TEXTLIST BetrAnzeigeListe
  6 = 'Einzel-Schritt, Litze einführen' | EN: 'Operating mode: Single step,  Steps with Start button, Exit with Single step' | DE: 'Betriebsart: Einzelschritt, Schritte mit Taste START, Beenden mit Einzelschritt' | FR: 'Mode de fonctionnement : Etape individuelle, Etape avec touche Start, Terminer avec étape individuelle' | HU: 'Üzemmód: Egyes lépés,  lépések a Start gombbal,  Befejezés egyes lépéssel' | IT: 'Modalità operativa: Passo-passo,  Avanzare con START, Uscire con Passo-passo' | RU: 'Режим работы: Отдельный шаг,  Шаги с кнопкой Start, ' | RO: 'Mod de operare: pas cu pas \\pasi cu tasta START\\ Iesire din "pas cu pas"' | ES: 'Modo de funcionamiento: Paso individual,  Pasos pulsando Start,  Salir con Paso individual' | PL: 'Tryb pracy: Pojedynczy krok,  Kroki poprzez przyscisk Start, Wyjście poprzez pojedynczy krok' | JA: '作業モード:\u3000シングルステップ, スタートボタンでステップ毎に動作, シングルステップの終了' | ZH: '运行模式: 步进模式, 按启动按钮步进, 通过步进退出'
  7 = 'Einzel-Schritt weiter mit Start' | EN: 'Operating mode: Single step  Steps with Start button Exit with Single step' | DE: 'Betriebsart: Einzelschritt, Schritte mit Taste START, Beenden mit Einzelschritt' | FR: 'Mode de fonctionnement : Etape individuelle Etape avec touche Start Terminer avec étape individuelle' | HU: 'Üzemmód: Egyes lépés  lépések a Start gombbal  Befejezés egyes lépéssel' | IT: 'Modalità operativa: Passo-passo  Avanzare con START Uscire con Passo-passo' | RU: 'Режим работы: Отдельный шаг  Шаги с кнопкой Start ' | RO: 'Mod de operare: pas cu pas \\pasi cu tasta START\\ Iesire din "pas cu pas"' | ES: 'Modo de funcionamiento: Paso individual  Pasos pulsando Start  Salir con Paso individual' | PL: 'Tryb pracy: Pojedynczy krok  Kroki poprzez przyscisk Start Wyjście poprzez pojedynczy krok' | JA: '作業モード:\u3000シングルステップ スタートボタンでステップ毎に動作 シングルステップの終了' | ZH: '运行模式: 步进模式 按启动按钮步进 通过步进退出'
  10 = 'Maschine bereit, Weiter mit Taste START' | EN: 'Machine ready  Continue with START button' | DE: 'Maschine bereit, Weiter mit Taste START' | FR: ' Machine opérationnelle  Continuer avec touche START' | HU: ' Gép készen áll  Tovább a START gombbal' | IT: 'Macchina pronta Premere il tasto START per continuare' | RU: 'Аппарат готов  Продолжить кнопкой START' | RO: 'Masina pregatita\\ Continua cu tasta START' | ES: 'Máquina preparada  Continue pulsando START' | PL: 'Maszyna gotowa  kontynuacja poprzez przycisk START' | JA: '準備完了\\スタートボタンを押してください' | ZH: ' 设备待机  按启动按钮继续'
  11 = 'Maschine bereit zum Crimpen - Litze einführen' | EN: 'Machine ready for crimping   Insert wire' | DE: 'Maschine bereit zum Crimpen, Litze einführen' | FR: 'Machine opérationnelle pour sertissage  Introduire fil' | HU: 'Gép krimpelésre kész  Huzal behelyezése\\' | IT: 'Macchina pronta per crimpare  Inserire il cavo' | RU: 'Машина готова к обжиму  Завести провод' | RO: 'Masina pregatita pentru sertizare\\ Introduceti lita' | ES: 'Máquina preparada para engaste   Insertar cable' | PL: 'Maszyna gotowa do zaciskania   Wprowadzić przewód' | JA: '圧着準備完了 ケーブル挿入' | ZH: '设备待机准备压接   送线'
  12 = 'Maschine im Ablauf gestoppt - Weiter mit START' | EN: 'Machine stopped during process  Continue with START' | DE: 'Maschine im Ablauf gestoppt, Weiter mit START' | FR: ' Machine arrêtée en cours  Continuer avec touche START' | HU: ' Gép a folyamat közben megállítva  Tovább a START-tal' | IT: 'La macchina si è bloccata durante il processo Premere START per continuare' | RU: 'Остановка машины во время работы  Продолжить кнопкой START' | RO: 'Masina s-a oprit in timpul procesului\\ Continua cu tasta START' | ES: 'Máquina parada durante el proceso  Continue con START' | PL: 'Maszyna zatrzymana w czasie procesu  kontynuacja poprzez przycisk START' | JA: '機械が動作中停止しました スタートボタンを押してください' | ZH: ' 运行中设备停止  按启动按钮继续'
  13 = 'nicht Crimpen zu (?)' | EN: 'Open crimping tool for setup Close with Start button Exit with Reset' | DE: 'Crimpzange zum Einrichten offen, Schließen mit Taste Start, Beenden mit Reset' | FR: 'Ouvrir pince à sertir pour réglage Fermer avec touche Start Terminer avec Reset' | HU: 'Krimpelo fogó beállításhoz nyitva  Zárás a Start gombbal  Befejezés a Reset gombbal' | IT: 'Apertura ganasce di crimpatura per regolazione Chiusura con pulsante START Uscire con RESET' | RU: 'Открыть обжимной элемент для настройки   Закрыть кнопкой Start  Выход через Reset' | RO: 'Cleste crimpare deschis pentru reglare\\ Inchidere cu tasta START\\ Incheiere cu tasta RESET' | ES: 'Herramienta de crimpado abierta para ajuste Cerrar pulsando Start Salir pulsando Reset' | PL: 'Otwarcie jednostki zaciskającej do ustawienia Zamknięcie poprzez przycisk Start Wyjście poprzez przycisk Reset' | JA: 'セットアップ時の圧着ツールオープン スタートボタンでクローズ/nリセッットで終了' | ZH: '打开压接工具来设定 按启动按钮关闭 按复位按钮退出'
  14 = 'Crimpen zu (?)' | EN: 'Crimping tool closed for testing Open with Start button Exit with Reset' | DE: 'Crimpzange zum Prüfen zu Öffnen mit Taste Start, Beenden mit Reset' | FR: 'Fermer pince à sertir pour contrôle Ouvrir avec touche Start Terminer avec Reset' | HU: 'Krimpelo fogó ellenorzéshez zárva  Nyitás a Start gombbal  Befejezés a Reset gombbal' | IT: 'Ganasce di crimpatura chiuse per test Aprire con pulsante START Uscire con RESET' | RU: 'Обжимной элемент закрыт для теста  Открыть кнопкой Старт Завершить с помощью Reset' | RO: 'Cleste crimpare inchis pentru verificare\\ deschidere cu tasta START\\ Incheiere  cu tasta RESET' | ES: 'Herramienta de crimpado cerrada para ajuste Abrir pulsando Start Salir pulsando Reset' | PL: 'Jednostka zaciskająca zamknięta do testowania Otwarcie maszyny poprzez przycisk Wyjście poprzez przycisk Reset' | JA: 'テスト時の圧着ツールクローズ スタートボタンでオープン リセットで終了' | ZH: '关闭压接工具来测试 按启动按钮开机 按复位按钮退出'
  15 = 'Bereit zum Crimpen - Litze einführen-dann Start drücken' | EN: 'Machine ready for crimping  Insert wire and press Start button' | DE: 'Maschine bereit zum Crimpen, Litze einführen und Taste Start drücken' | FR: 'Machine opérationnelle pour sertissage  Introduire fil et appuyer touche Start' | HU: 'Gép krimpelésre kész  Huzal behelyezése\\ és  nyomja meg a Start gombot' | IT: 'Macchina pronta per crimpare Inserire il cavo e premere il pulsante START' | RU: 'Машина готова к обжиму  Завести провод и  нажать кнопку Старт' | RO: 'Masina pregatita pentru sertizare\\ Introduceti lita si \\ apasa tasta START' | ES: 'Máquina preparada para engaste  Insertar cable y pulsar Start' | PL: 'Maszyna gotowa do zaciskania  Wprowadzić przewód i  nacisnąć przycisk Start' | JA: '圧着準備完了 ケーブル挿入 スタートボタンを押してください' | ZH: '设备待机准备压接  送线  按下启动按钮'
  20 = 'Abisolieren einrichten - weiter mit Start' | EN: 'Operating mode:  Set up stripping unit Continue with Start Exit with Reset' | DE: 'Betriebsart: Abisolieren einrichten, weiter mit Start, Beenden mit Reset' | FR: 'Mode de fonctionnement :  Régler dénudage Continuer avec Start Terminer avec Reset' | HU: 'Üzemmód:  Csupaszítás beállítása  tovább a Start gombbal Befejezés a Reset gombbal' | IT: 'Modalità operativa: Impostazione unità di spellatura Continuare con START Uscire con RESET' | RU: 'Режим работы: Настройка снятия изоляции  Продолжить с Start Выход с Reset' | RO: 'Mod de operare: reglare dezizolare\\continua cu tasta START\\ Incheiere cu RESET' | ES: 'Modo de funcionamiento: Ajustar unidad de pelado Continuar con Start Salir con Reset' | PL: 'Tryb pracy: Ustawianie jednostki zaciskającej Kontynuacja poprzez przycisk Start Wyjście poprzez przycisk Reset' | JA: '作業モード:\u3000ストリッピング・ユニットのセットアップ スタートして継続/リセットして終了' | ZH: '运行模式: 设定剥线单元  按启动按钮继续 通过复位退出 '
  21 = 'Magazin Leerfahren (?)' | EN: 'Operating mode:  Run magazine empty Exit with Reset' | DE: 'Betriebsart: Magazin leerfahren, Beenden mit Reset' | FR: 'Mode de fonctionnement :  Vider magasin Terminer avec Reset' | HU: 'Üzemmód:  Tároló üresre járatása Befejezés a Reset gombbal' | IT: 'Modalità operativa:  Svuotamento caricatore Uscire con RESET' | RU: 'Вид операции:  Очистить магазин Завершить с помощью Reset' | RO: 'Mod de operare: \\ golire magazie \\ Incheiere  cu tasta RESET' | ES: 'Modo de funcionamiento:  Ejecutar vaciado de depósito Salir con Reset' | PL: 'Tryb pracy:   Uruchomienie pustego magazynka Wyjście poprzez przycisk Reset' | JA: '作業モード:\u3000 マガジンが空の状態での操作 リセットで終了' | ZH: '运行模式:   启动料箱清空 通过复位退出 '
  22 = 'Sortierer Leerfahren (?)' | EN: 'Operating mode:  Run sorter empty Exit with Reset' | DE: 'Betriebsart: Sortierer leerfahren, Beenden mit Reset' | FR: 'Mode de fonctionnement :  Vider trieuse Terminer avec Reset' | HU: 'Üzemmód:  Szortírozó üresre járatása Befejezés a Reset gombbal' | IT: 'Modalità operativa: Scarico canale contatti Uscire con RESET' | RU: 'Вид операции:  Очистка сортировщика Завершить с помощью Reset' | RO: 'Mod de operare: \\ golire sortator \\ Incheiere  cu tasta RESET' | ES: 'Modo de funcionamiento:  Ejecutar vaciado clasificador Salir con Reset' | PL: 'Tryb pracy:   Uruchomienie pustego sortera Wyjście poprzez przycisk Reset' | JA: '作業モード:\u3000 ソーター空状態での操作 リセットで終了' | ZH: '运行模式:   运行分拣清空 通过复位退出 '
  23 = 'Crimpen Einrichten (?)' | EN: 'Operating mode:  Set up crimping Exit with Reset' | DE: 'Betriebsart: Crimpzange einrichten, Beenden mit Reset' | FR: 'Mode de fonctionnement :  Régler pince à sertir Terminer avec Reset' | HU: 'Üzemmód:  Krimpelo fogó beállítása Befejezés a Reset gombbal' | IT: 'Modalità operativa:  Regolazione crimpatura Uscire con RESET' | RU: 'Вид операции:  Настройка обжимного элемента Завершить с помощью Reset' | RO: 'Mod de operare: \\ reglare cleste sertizare\\ Incheiere cu tasta RESET' | ES: 'Modo de funcionamiento:  Ajustar engaste Salir con Reset' | PL: 'Tryb pracy:   Ustawienie zaciskania Wyjście poprzez przycisk Reset' | JA: '作業モード:\u3000 圧着の設定 リセットで終了' | ZH: '运行模式:   设定压接 通过复位退出 '
  24 = 'Abisolieren einrichten - Litze einführen' | EN: 'Operating mode:  Set up stripping unit Insert wire Exit with Reset' | DE: 'Betriebsart: Abisolieren einrichten, Litze einführen, Beenden mit Reset' | FR: 'Mode de fonctionnement :  Régler dénudage Introduire fil Terminer avec Reset' | HU: 'Üzemmód:  Csupaszítás beállítása Huzal behelyezése Befejezés a Reset gombbal' | IT: 'Modalità operativa: Impostazione unità di spellatura Inserire il cavo Uscire con RESET' | RU: 'Режим работы: Настройка снятия изоляции  завести провод Выход с Reset' | RO: 'Mod de operare: reglare dezizolare\\ introducere lita\\ Incheiere cu RESET' | ES: 'Modo de funcionamiento: Ajustar unidad de pelado Insertar cable Salir con Reset' | PL: 'Tryb pracy: Ustawianie jednostki zaciskającej Wprowadzić przewód Wyjście poprzez przycisk Reset' | JA: '作業モード:\u3000ストリッピング・ユニットのセットアップ ケーブルの挿入/リセットして終了' | ZH: '运行模式: 设定剥线单元   送线   通过复位退出 '
  25 = 'Probelauf ohne Kontakt' | EN: 'Operating mode:  Trial run without contact Exit with Reset' | DE: 'Betriebsart: Probelauf ohne Kontakt, Beenden mit Reset' | FR: "Mode de fonctionnement :  Marche d'essai sans contact Terminer avec Reset" | HU: 'Üzemmód:  Próbaüzem érintkezo nélkül Befejezés a Reset gombbal' | IT: 'Modalità operativa: Ciclo di prova senza contatto Uscire con RESET' | RU: 'Вид операции:  Пробный запуск без контактов Завершить с помощью Reset' | RO: 'Mod de operare: \\ test fara contacte \\ Incheiere  cu tasta RESET' | ES: 'Modo de funcionamiento:  Prueba sin contacto  Salir con Reset' | PL: 'Tryb pracy:   Przebieg testowy bez kontaktu Wyjście poprzez przycisk Reset' | JA: '作業モード:\u3000 コンタクトなしでのテスト操作 リセットで終了' | ZH: '运行模式:   试运行但不进针 通过复位退出 '
  26 = 'Probelauf ohne Crimpen' | EN: 'Operating mode:  Trial run without crimping Exit with Reset' | DE: 'Betriebsart: Probelauf ohne Crimpen, Beenden mit Reset' | FR: "Mode de fonctionnement :  Marche d'essai sans sertissage Terminer avec Reset" | HU: 'Üzemmód:  Próbaüzem krimplelés nélkül Befejezés a Reset gombbal' | IT: 'Modalità operativa: Ciclo di prova senza crimpatura Uscire con RESET' | RU: 'Вид операции:  Пробный запуск без обжима Завершить с помощью Reset' | RO: 'Mod de operare: \\ test fara sertizare \\ Incheiere  cu tasta RESET' | ES: 'Modo de funcionamiento:  Prueba sin engaste  Salir con Reset' | PL: 'Tryb pracy:   Przebieg testowy bez zaciskania Wyjście poprzez przycisk Reset' | JA: '作業モード:\u3000 圧着なしでのテスト操作 リセットで終了' | ZH: '运行模式:   试运行但不压接 通过复位退出 '
  27 = 'Probelauf ohne Litze' | EN: 'Operating mode:  Trial run without wire Exit with Reset' | DE: 'Betriebsart: Probelauf ohne Litze Beenden, mit Reset' | FR: "Mode de fonctionnement :  Marche d'essai sans fil Terminer avec Reset" | HU: 'Üzemmód:  Próbaüzem huzal nélkül Befejezés a Reset gombbal' | IT: 'Modalità operativa: Ciclo di prova senza cavo Uscire con RESET' | RU: 'Вид операции:  Пробный запуск без кабеля Завершить с помощью Reset' | RO: 'Mod de operare: \\ test fara lite \\ Incheiere cu tasta RESET' | ES: 'Modo de funcionamiento:  Prueba sin cable  Salir con Reset' | PL: 'Tryb pracy:   Przebieg testowy bez przewodu Wyjście poprzez przycisk Reset' | JA: '作業モード:\u3000 ケーブルなしでのテスト操作 リセットで終了' | ZH: '运行模式:   试运行但不进线 通过复位退出 '
  55 = 'A55 Kontakt nicht gefallen' | EN: 'Malfunction: Contact not fed E1.10 missing' | DE: 'Störung: Kontakt nicht gefallen E1.10 fehlt' | FR: 'Défaut : contact pas tombé E1.10 absent' | HU: 'Zavar: Érintkezo nem esett le E1.10 hiányzik' | IT: 'Anomalia: Contatto non in posizione E1.10 mancante' | RU: 'Нарушение: Контакт не загружен, E1.10 отсутствует' | RO: 'Defectiune: Contactul nu a cazut\\ E1.10 lipseste' | ES: 'Error de funcionamiento: Contactos no alimentados E1.10 sin señal' | PL: 'Nieprawidłowość:  Kontakt niepodany E1.10 Brakuje' | JA: 'エラー: コンタクトが供給されていません E1.10\u3000不明' | ZH: '故障: 针没有落下 E1.10 故障'
  1000 = 'ohne Sortierluft' | EN: 'without sorting air' | DE: 'ohne Sortierluft' | FR: "sans tri d'air" | HU: 'buborékok nélkül' | IT: 'senza aria' | RU: 'без пузырьков' | RO: 'fără bule' | ES: 'sin burbujas' | PL: 'bez bąbelków' | JA: '空気をソートせずに' | ZH: '没有分拣气'
  1001 = 'mit Sortierluft' | EN: 'with sorting air' | DE: 'mit Sortierluft' | FR: "avec tri de l'air" | HU: 'buborékokkal' | IT: 'con aria' | RU: 'с пузырьками' | RO: 'cu bule' | ES: 'con burbujas' | PL: 'z bąbelkami' | JA: 'ソートエアー付き' | ZH: '带分拣气'
  127 = 'warte auf SAFETY-Signal...'
  101 = 'Druckluft nicht ein'
  102 = 'Schutztür nicht zu'
  105 = 'Kein Signal von Taste Maschine-Aus'
  108 = 'Not-Aus Steuerpult nicht OK'
  109 = 'Kein SAFETY Signal'
  501 = 'Fehler: A1.8 "Kontakt schieben" ist aus, aber Schieber ist vorn.'
  502 = 'Fehler: A1.8 "Kontakt schieben" ist ein, aber Schieber ist nicht vorn.'
  503 = 'Fehler: A1.9 "Crimpeinheit vor" ist aus, Einheit ist aber nicht hinten.'
  504 = 'Fehler: A1.9 "Crimpeinheit vor" ist ein, Einheit ist aber nicht vorn.'
  505 = 'Fehler: A1.10 "Abisolierer nach links" ist aus, aber Einheit ist links.'
  506 = 'Fehler: A1.10 "Abisolierer nach links" ist ein, aber Einheit ist nicht links.'
  507 = 'Fehler: A1.11 "Abisolierer zu" ist aus, aber Abisolierer ist zu.'
  508 = 'Fehler: A1.11 "Abisolierer zu" ist ein, aber Abisolierer ist nicht zu.'
  509 = 'Fehler A1.13 "Abisolierer zurück" ist aus, aber Abisolierer ist nicht vorn.'
  510 = 'Fehler A1.13 "Abisolierer zurück" ist ein, aber Abisolierer ist nicht hinten.'
  511 = 'Fehler A1.14 "Crimpzange zu" ist aus, aber Zange ist nicht offen.'
  512 = 'Fehler A1.14 "Crimpzange zu" ist ein, aber Zange ist offen.'
  513 = 'Fehler A1.15 "Drahthalter zu" ist aus, aber Drahthalter ist nicht offen.'
  514 = 'Fehler A1.15 "Drahthalter zu" ist ein, aber Drahthalter ist offen.'
  500 = '   '
  420 = 'Einzelschritt - Start durch Drahteinfuhr'
  422 = 'Abisolierer zu'
  423 = 'Abisolierer zurück (abisolieren)'
  424 = 'Abisolierer nach links + Abisolierer auf'
  425 = 'Crimpeinheit vor'
  426 = 'Crimpen zu'
  427 = 'Drahthalter + Drahtführung auf'
  428 = 'Crimpzange auf + Abisoliereinheit vor'
  429 = 'Ausstoßen vor'
  430 = 'Crimpeinheit zurück'
  431 = 'Abisolierer nach rechts + Kontakt-Schieben zurück'
  432 = 'Einzelschritt - Ende'
  421 = 'Drahthalter + Drahtführung zu'
  600 = 'Störung: Drahthalter nicht offen, E1.2 fehlt' | EN: 'Malfunction: Wire holder not open, E1.2 missing' | DE: 'Störung: Drahthalter nicht offen, E1.2 fehlt' | FR: 'Défaut : Porte-fil pas ouvert, E1.2 absent' | HU: 'Zavar: Huzaltartó nincs nyitva, E1.2 hiányzik' | IT: 'Anomalia: Dispositivo blocca-cavo chiuso, E1.2 mancante' | RU: 'Нарушение: Кабельный захват не открыт, E1.2 отсутствует' | RO: 'Defectiune: Suportul de fir nu e deschis, E1.2 lipseste' | ES: 'Error de funcion.: Soporte de cable no está abierto, E1.2 sin señal' | PL: 'Nieprawidłowość: Uchwyt przewodu nie jest otwarty, E1.2 Brakuje' | JA: 'エラー: ケーブルフォルダーが閉じていません, E1.2 不明' | ZH: '故障: 集线器未打开, E1.2 缺失'
  601 = 'Störung: Drahthalter nicht zu E1.2 nicht weg' | EN: 'Malfunction: Wire holder not closed, E1.2 not gone' | DE: 'Störung: Drahthalter nicht zu, E1.2 nicht weg' | FR: 'Défaut : Porte-fil pas fermé, E1.2 pas parti' | HU: 'Zavar: Huzaltartó nincs zárva, E1.2 nem tunt el' | IT: 'Anomalia: Dispositivo blocca-cavo aperto, E1.2 non attivo' | RU: 'Нарушение: Кабельный захват не закрыт, E1.2 не удален' | RO: 'Defectiune: Suportul de fir nu e inchis, E1.2 nu dispare' | ES: 'Error de funcion.: Soporte de cable no está cerrado, E1.2 no desaparece la señal' | PL: 'Nieprawidłowość: Uchwyt przewodu nie jest zamknięty, E1.2 Pozostaje' | JA: 'エラー: ワイヤーホルダーが閉じていません, E1.2 不明' | ZH: '故障: 集线器未关闭, E1.2 没有离开'
  602 = 'Störung: Auslöseschalter Dauermeldung E1.3 nicht weg' | EN: 'Malfunction: Cable trigger switch continuous signal, E1.3 not gone' | DE: 'Störung: Auslöseschalter Dauermeldung, E1.3 nicht weg' | FR: 'Défaut : Déclencheur message permanent, E1.3 pas parti' | HU: 'Zavar: Kioldó kapcsoló folyamatos jelzés, E1.3 nem tunt el' | IT: 'Anomalia: Segnale continuo del sensore di presenza cavo, E1.3 non attivo' | RU: 'Нарушение: Непрерывный сигнал блокировки, E1.3 не удален' | RO: 'Defectiune: Declanșator mesaj permanent, E1.3 nu dispare' | ES: 'Error de funcion.: Señal permanente en interruptor de disparo de cable, E1.3 no desaparece' | PL: 'Nieprawidłowość: Przełącznik kablowy z ciągłym sygnałem, E.1.3 Pozostało' | JA: 'エラー: ケーブルトリガースイッチが連続メッセージ, E1.3\u3000未完了' | ZH: '故障:线缆触发开关持续信号, E1.3 故障没有解除'
  603 = 'Störung: Abisoliermesser nicht offen E1.4 nicht weg' | EN: 'Malfunction: Stripping blades not open, E1.4 not gone' | DE: 'Störung: Abisoliermesser nicht offen, E1.4 nicht weg' | FR: 'Défaut : Lames à dénuder pas ouvertes, E1.4 pas parti' | HU: 'Zavar: Csupaszító kés nincs nyitva, E1.4 nem  tunt el' | IT: 'Anomalia: Lame di spellatura non aperte, E1.4 non attivo' | RU: 'Нарушение: Нож зачистки не открыт, E1.4 не удален' | RO: 'Defectiune: Cutitul de dezizolare nu e deschis, E1.4 nu dispare' | ES: 'Error de funcion.: Cuchillas de pelado no abiertas, E1.4 no desaparece la señal' | PL: 'Nieprawidłowość:  Noże odizolowujące nie są otwarte, E1.4 Pozostało' | JA: 'エラー: ストリッピングブレードが開いていません,  E1.4\u3000未完了' | ZH: '故障: 剥线刀片没有打开, E1.4 故障没有解除'
  604 = 'Störung: Abisoliermesser nicht  zu E1.4 fehlt' | EN: 'Malfunction: Stripping blades not closed, E1.4 missing' | DE: 'Störung: Abisoliermesser nicht  zu, E1.4 fehlt' | FR: 'Défaut : Lames à dénuder pas fermées, E1.4 absent' | HU: 'Zavar: Csupaszító kés nincs zárva, E1.4 hiányzik' | IT: 'Anomalia: Lame di spellatura non chiuse, E1.2 mancante' | RU: 'Нарушение: Нож зачистки не закрыт, E1.4 отсутствует' | RO: 'Defectiune: Cutitul de dezizolare nu e inchis, E1.4 lipseste' | ES: 'Error de funcion.: Cuchillas de pelado no cerradas, E1.4 sin señal' | PL: 'Nieprawidłowość: Nnoże odizolowujące nie są zamknięte, E1.4 Brakuje' | JA: 'エラー: ストリッピングブレードが閉じていません, 1.4不明' | ZH: '故障: 剥线刀片没有闭合 E1.4 故障'
  605 = 'Störung: Doppelmeldung Abisolierer vorn+rück E1.5+E1.6 gleichzeitig' | EN: 'Malfunction: Double signal stripping unit at front+rear E1.5+E1.6 simultaneous' | DE: 'Störung: Doppelmeldung Abisolierer vorn+rück, E1.5+E1.6 gleichzeitig' | FR: 'Défaut : Message double Dénudeur avance+retour, E1.5+E1.5 simultanément' | HU: 'Zavar: Dupla jelzés Csupaszító elol+vissza, E1.5+E1.6 egyszerre' | IT: 'Anomalia: Segnale doppio Unità di spellatura avanzata+arretrata E1.5+E1.6 contemporaneamente' | RU: 'Нарушение: Двухкратное сообщение блок зачистки фронтальный + задней панелиnE1.3+E1.4 одновременно' | RO: 'Defectiune: Mesaj dublu dezizolator inainte+inapoi, E1.5+E1.6 simultan' | ES: 'Error de funcion.: Doble señal la unidad de pelado está delante y detrás E1.3+E1.4 simultaneamente' | PL: 'Nieprawidłowość: Podwójny sygnał jednostka odizolowująca z przodu+tyłu E1.3+E1.4 Równocześnie' | JA: 'エラー:ダブルメッセージ ストリッピングユニットが前面+後方にあります E2.1+E2.4\u3000同時発生' | ZH: '故障:    双路信号 剥线单元在前+在后 E1.3+E1.4 同时'
  606 = 'Störung: Abisolierer nicht vorn E1.5 fehlt' | EN: 'Malfunction: Stripping unit not at front, E1.5 missing' | DE: 'Störung: Abisolierer nicht vorn, E1.5 fehlt' | FR: 'Défaut : Dénudeur pas avance, E1.5 absent' | HU: 'Zavar: Csupaszító kés nincs elöl, E1.5 hiányzik' | IT: 'Anomalia: Unità di spellatura non avanzata, E1.5 mancante' | RU: 'Нарушение: Зачистка не фронтально, E1.5 отсутствует' | RO: 'Defectiune: Dezizolatorul nu e in fata, E1.5 lipseste' | ES: 'Error de funcion.: La unidad de pelado no está en la parte frontal, E1.3 sin señal' | PL: 'Nieprawidłowość: Jednostka odizolowująca nie jest z przodu, E1.5 Brakuje' | JA: 'エラー: ストリッピングユニットが前面に有りません, E1.5\u3000不明' | ZH: '故障: 剥线单元不在前边, E1.5 故障'
  607 = 'Störung: Abisolierer nicht rück (abisoliert) E1.6 fehlt' | EN: 'Malfunction: Stripping unit not at rear (stripped),  E1.6 missing' | DE: 'Störung: Abisolierer nicht rück (abisoliert),  E1.6 fehlt' | FR: 'Défaut : Dénudeur pas retour (dénudé),  E1.6 absent' | HU: 'Zavar: Csupaszító nincs hátul (csupaszított), E1.6 hiányzik' | IT: 'Anomalia: Unità si spellatura non arretrata (spellato), E1.6 mancante' | RU: 'Нарушение: Зачистка не с тыльной стороны (зачистка), E1.6 отсутствует' | RO: 'Defectiune: Dezizolatorul nu revine in spate, E1.6 lipseste' | ES: 'Error de funcion.: La unidad de pelado no está en la parte posterior (despojado), E1.6 sin señal' | PL: 'Nieprawidłowość: Jednostka odizolowująca nie jest z tyłu (odizolowane), E1.6 Brakuje' | JA: 'エラー: ストリッピングユニットが後方に有りません （除去済み), E1.6 不明' | ZH: '故障: 剥线单元不在后边 (剥离), E1.6 故障'
  608 = 'Störung: Abisolierer nicht links (aus Arbeitsraum) E1.7 fehlt' | EN: 'Malfunction: Stripping unit not on LH side (out of machining compartment), E1.7 missing' | DE: 'Störung: Abisolierer nicht links (aus Arbeitsraum), E1.7 fehlt' | FR: "Défaut : Dénudeur pas gauche (de l'espace de travail), E1.7 absent" | HU: 'Zavar: Csupaszító nincs bal oldalon (a munkatérbol), E1.7 hiányzik' | IT: 'Anomalia: Unità di spellatura non sul lato LH (fuori dal comparto di lavoro), E1.7 mancante' | RU: 'Нарушение: Блокзачистки не с лева (вне машинного блока), E1.7 отсутствует' | RO: 'Defectiune: Dezizolatorul nu e in stanga (din domeniul de lucru), E1.7 lipseste' | ES: 'Error de funcion.: La unidad de pelado no está en el lado LH (fuera del espacio de trabajo), E1.7 sin señal' | PL: 'Nieprawidłowość: Jednostka odizolowująca nie jest z lewej strony (poza przedziałem maszyny), E1.7 Brakuje' | JA: 'エラー: ストリッピングユニットがLH側に有りません (正しくセットされていません）E1.7 不明' | ZH: '故障: 剥线单元不在左边 ( 不在工作区间 )  E1.7 故障'
  609 = 'Störung: Abisolierer nicht rechts E1.7 nicht weg' | EN: 'Malfunction: Stripping unit not on RH side, E1.7 not gone' | DE: 'Störung: Abisolierer nicht rechts, E1.7 nicht weg' | FR: 'Défaut : Dénudeur pas droite, E1.7 pas parti' | HU: 'Zavar: Huzaltartó nincs jobb oldalon, E1.7 nem tunt el' | IT: 'Anomalia: Unità di spellatura non sul lato RH, E1.7 non attivo' | RU: 'Нарушение: Блокзачистки не с права, E1.7 не удален' | RO: 'Defectiune: Dezizolatorul nu e in dreapta, E1.7 nu dispare' | ES: 'Error de funcionamiento: La unidad de pelado no está en el lado RH, E1.7 no desaparece la señal' | PL: 'Nieprawidłowość: Jednostka odizolowująca nie jest po prawej stronie, E1.7 Pozostało' | JA: 'エラー: ストリッピングユニットがRH側に有りません E1.5\u3000未完了' | ZH: '故障: 剥线单元不在右边, E1.7 故障没有解除'
  610 = 'Störung: Doppelmeldung Crimpzange zu+offen E1.8+E1.9 gleichzeitig' | EN: 'Malfunction: Double signal Crimping tool closed+open, E1.8+E1.9 simultaneous' | DE: 'Störung: Doppelmeldung Crimpzange zu+offen E1.8+E1.9 gleichzeitig' | FR: 'Défaut : Message double Pince à sertir fermée+ouverte E1.8+E1.9 simultanément' | HU: 'Zavar: Dupla jelzés Krimpelo fogó zárva+nyitva, E1.8+E1.9 egyszerre' | IT: 'Anomalia: Segnale doppio Ganasce di crimpatura chiuse+aperte, E1.8+E1.9 contemporaneamente' | RU: 'Нарушение: Двухкратное сообщение обжимной элемент закрать + открыть, E1.8+E1.9 одновременно' | RO: 'Defectiune: Mesaj dublu cleste sertizare inchis+deschis, E1.8+E1.9 simultan' | ES: 'Error de funcionamiento: Doble señal la unidad de crimpado está abierta y cerrada, E1.8+E1.9 simultaneamente' | PL: 'Nieprawidłowość: Podwójny sygnał Jednostka zaciskająca zamknięta+otwarta, E1.8+E1.9 Równocześnie' | JA: 'エラー:ダブルメッセージ ストリッピングユニット\u3000クローズ+オープン E1.8+E1.9 同時発生' | ZH: '故障:   双路信号 压接工具闭合+打开 E1.8+E1.9 同时'
  611 = 'Störung: Crimpzange nicht zu E1.8 fehlt' | EN: 'Malfunction: Crimping tool not closed, E1.8 missing' | DE: 'Störung: Crimpzange nicht zu, E1.8 fehlt' | FR: 'Défaut : Pince à sertir pas fermée, E1.8 absent' | HU: 'Zavar: Csupaszító kés nincs zárva E1.8 hiányzik' | IT: 'Anomalia: Ganasce di crimpatura aperte, E1.8 mancante' | RU: 'Нарушение: Обжимной элемент не закрыт, E1.8 отсутствует' | RO: 'Defectiune: Clestele de sertizare nu e inchis, E1.8 lipseste' | ES: 'Error de funcionamiento: Herramienta de engaste no está cerrada, E1.8 sin señal' | PL: 'Nieprawidłowość: Jednostka zaciskająca nie jest zamknięta, E1.8 Brakuje' | JA: 'エラー: 圧着ツールが閉じていませんE1.8\u3000不明' | ZH: '故障: 压接工具没有关闭, E1.8 故障'
  612 = 'Störung: Crimpzange nicht offen E1.7 fehlt' | EN: 'Malfunction: Crimping tool not open, E1.9 missing' | DE: 'Störung: Crimpzange nicht offen, E1.9 fehlt' | FR: 'Défaut : Pince à sertir pas ouverte, E1.9 absent' | HU: 'Zavar: Csupaszító kés nincs nyitva E1.9 hiányzik' | IT: 'Anomalia: Ganasce di crimpatura chiuse E1.9 mancante' | RU: 'Нарушение: Обжимной элемент не открыт, E1.9 отсутствует' | RO: 'Defectiune: Clestele de sertizare nu e deschis, E1.9 lipseste' | ES: 'Error de funcionamiento: Herramienta de engaste no está abierta, E1.9 sin señal' | PL: 'Nieprawidłowość: Jednostka zaciskająca nie jest otwarta, E1.9 Brakuje' | JA: 'エラー: 圧着ユニットが開いていません, E1.9 不明' | ZH: '故障: 压接工具没有打开, E1.9 故障'
  613 = 'Störung: Kontakt nicht gefallen E1.10 fehlt' | EN: 'Malfunction: Contact not fed, E1.10 missing' | DE: 'Störung: Kontakt nicht gefallen, E1.10 fehlt' | FR: 'Défaut : Contact pas tombé, E1.10 absent' | HU: 'Zavar: Érintkezo nem esett le, E1.10 hiányzik' | IT: 'Anomalia: Contatto non in posizione E1.10 mancante' | RU: 'Нарушение: Контакт не загружен, E1.10 отсутствует' | RO: 'Defectiune: Contactul nu a cazut E1.10 lipseste' | ES: 'Error de funcion.: Contactos no alimentados, E1.10 sin señal' | PL: 'Nieprawidłowość: Kontakt niepodany, E1.10 Brakuje' | JA: 'エラー: コンタクトが供給されていません 1.10\u3000不明' | ZH: '故障: 针没有落下 E1.10 故障'
  614 = 'Störung: Dauermeldung Kontakt gefallen E1.10 nicht weg' | EN: 'Malfunction: Continuous signal, contact fed, E1.10 not gone' | DE: 'Störung: Dauermeldung Kontakt gefallen, E1.10 nicht weg' | FR: 'Défaut : Message permanent contact tombé, E1.10 pas parti' | HU: 'Zavar: Folyamatos jelzés érintkezo leesett, E1.10 nem tunt el' | IT: 'Anomalia: Segnale continuo alimentatore dei contatti, E1.10 non attivo' | RU: 'Нарушение: Непрерывный сигнал контакт не загружен, E1.10 не удален' | RO: 'Defectiune: Mesaj permanent contact cazut, E1.10 nu dispare' | ES: 'Error de funcionamiento: Señal permanente alimentador contactos, E1.10 no desaparece la señal' | PL: 'Nieprawidłowość: Ciągły sygnał, podajnik kontaktów E1.10 Pozostaje' | JA: 'エラー: 連続メッセージ,コンタクト供給, E1.10 未完了' | ZH: '故障: 持续信号，送针, E1.10 故障没有解除'
  615 = 'Störung: Doppelmeldung Crimpeinheit vorn+rück E1.11+E1.12 gleichzeitig' | EN: 'Malfunction:  Double signal Crimping unit at front+rear, E1.11+E1.12 simultaneous' | DE: 'Störung: Doppelmeldung Crimpeinheit vorn+rück, E1.11+E1.12 gleichzeitig' | FR: 'Défaut : Message double Unité à dénuder avance+retour, E1.11+E1.12 simultanément' | HU: 'Zavar:  Dupla jelzés Krimpelo egység elöl+hátul, E1.11+E1.12 egyszerre' | IT: 'Anomalia: Segnale doppio Unità di crimpatura avanzata+arretrata, E1.11+E1.12 contemporaneamente' | RU: 'Нарушение: Двухкратное сообщение Обжимной элемент фронтальный+задний, E1.11+E1.12  одновременно' | RO: 'Defectiune: mesaj dublu unitate sertizare inainte+inapoi E1.11+E1.12 simultan' | ES: 'Error de funcionamiento: Doble señal la unidad de crimpado está delante y detrás E1.11+E1.12 simultaneamente' | PL: 'Nieprawidłowość: Podwójny sygnał Jednostka zaciskająca z przodu+tyłu, E1.11+E1.12 Równocześnie' | JA: 'エラー:ダブルメッセージ 圧着ユニットが前面+後方にありません E1.11+E1.12 同時発生' | ZH: '故障:  双路信号 压接单元 在前+在后 E1.11+E1.12 同时'
  616 = 'Störung: Crimpeinheit nicht vorn E1.11 fehlt' | EN: 'Malfunction: Crimping unit not at front, E1.11 missing' | DE: 'Störung: Crimpeinheit nicht vorn, E1.11 fehlt' | FR: 'Défaut : Unité à dénuder pas avance, E1.11 absent' | HU: 'Zavar: Krimpelo egység nincs elöl, E1.11 hiányzik' | IT: 'Anomalia: Unità di crimpatura non avanzata, E1.11 mancante' | RU: 'Нарушение: Обжимной элемент не фронтально, E1.11 отсутствует' | RO: 'Defectiune: Unitatea de sertizare nu e in fata, E1.11 lipseste' | ES: 'Error de funcionamiento: Unidad de engaste no está en la parte frontal, E1.11 sin señal' | PL: 'Nieprawidłowość: Jednostka zaciskająca nie jest z przodu, E1.11 Brakuje' | JA: 'エラー: 圧着ユニットが前面に有りません,E1.11 不明' | ZH: '故障: 压接单元不在前面 E1.11 故障'
  617 = 'Störung: Crimpeinheit nicht rück E1.12 fehlt' | EN: 'Malfunction: Crimping unit not at rear, E1.12 missing' | DE: 'Störung: Crimpeinheit nicht rück, E1.12 fehlt' | FR: 'Défaut : Unité à dénuder pas retour, E1.12 absent' | HU: 'Zavar: Krimpelo egység nincs hátul, E1.12 hiányzik' | IT: 'Anomalia: Unità di crimpatura non arretrata E1.12 mancante' | RU: 'Нарушение: Обжимной элемент не с тыльной стороны, E1.12 отсутствует' | RO: 'Defectiune: Unitatea de sertizare nu e in spate E1.12 lipseste' | ES: 'Error de funcionamiento: Unidad de engaste no está en la parte posterior, E1.12 sin señal' | PL: 'Nieprawidłowość: Jednostka zaciskająca nie jest z tyłu E2.4 Brakuje' | JA: 'エラー: 圧着ユニットが後方に有りません E1.12\u3000不明' | ZH: '故障: 压接单元不在后面 E1.12 故障'
  618 = 'Störung: Kontakt-Schieben nicht vorn E1.14 fehlt' | EN: 'Malfunction: Contact slides not at front, E1.14 missing' | DE: 'Störung: Kontakt-Schieben nicht vorn, E1.14 fehlt' | FR: 'Défaut : Pousser contact pas avance, E1.14 absent' | HU: 'Zavar: Érintkezo-toló nincs elöl, E1.14 hiányzik' | IT: 'Anomalia. Slitta contatti non avanzata,  E1.14 mancante' | RU: 'Нарушение:  Контакт заведен не фронтально, E1.14 отсутствует' | RO: 'Defectiune: Impingatorul de contacte nu e in fata, E1.14 lipseste' | ES: 'Error de funcionamiento: Pasador de contactos no está en la parte frontal, E1.14 sin señal' | PL: 'Nieprawidłowość:  Zjeżdżalnia kontaktów nie jest z przodu,  E1.14 Brakuje' | JA: 'エラー: コンタクトスライドが前方に有りません E1.14 未装着 ' | ZH: '故障: 推针器在前面  E1.14 故障'
  619 = 'Störung: Kontakt-Schieben nicht rück E1.14 nicht weg' | EN: 'Malfunction: Contact slides not at rear E1.14 not gone' | DE: 'Störung: Kontakt-Schieben nicht rück, E1.14 nicht weg' | FR: 'Défaut : Pousser contact pas retour, E1.14 pas parti' | HU: 'Zavar: Érintlezo-toló nincs hátul, E1.14 nem tunt el' | IT: 'Anomalia. Slitta contatti non arretrata,  E1.14 non attivo' | RU: 'Нарушение:  Контакт заведен не с тыльной стороны, E1.14 не удален' | RO: 'Defectiune: Impingatorul de contacte nu e in spate, E1.14 nu dispare' | ES: 'Error de funcionamiento: Pasador de contactos no está en la parte posterior, E1.14 no desaparece la señal' | PL: 'Nieprawidłowość:  Zjeżdżalnia kontaktów nie jest z tyłu,  E1.14 Pozostaje' | JA: 'エラー: コンタクトスライドが後方に有りません E1.14\u3000未完了' | ZH: '故障: 推针器不在后面  E1.14 故障没有解除'
  620 = 'Störung: Ausstoßen nicht vorn E1.13 fehlt' | EN: 'Malfunction: Ejector not at front , E1.13 missing' | DE: 'Störung: Ausstoßen nicht vorn , E1.13 fehlt' | FR: 'Défaut : éjecter pas avance , E1.13 absent' | HU: 'Zavar: Kilökés nincs elöl , E1.13 hiányzik' | IT: 'Anomalia: Espulsore non avanzato , E1.13 mancante' | RU: 'Нарушение: Выталкивание не фронтальное , E1.13 отсутствует' | RO: 'Defectiune: Ejectorul nu e in fata\\ E2.3 lipseste' | ES: 'Error de funcionamiento: Eyector no está en la parte frontal , E1.13 sin señal' | PL: 'Nieprawidłowość:  Wyrzutnik nie jest z przodu .E2.3 Brakuje' | JA: 'エラー： エジェクタが前面に有りません 2.3\u3000未完了' | ZH: '故障: 弹射器不在前面 , E1.13 故障'
  621 = 'Störung: Ausstoßen nicht rück E1.13 nicht weg' | EN: 'Malfunction: Ejector not at rear , E1.13 not gone' | DE: 'Störung: Ausstoßen nicht rück , E1.13 nicht weg' | FR: 'Défaut : éjecter pas retour , E1.13 pas parti' | HU: 'Zavar: Kilökés nincs hátul , E1.13 nem tunt el' | IT: 'Anomalia: Espulsore non arretrato , E1.13 non attivo' | RU: 'Нарушение: Выталкивание не с тыльной стороны , E1.13 не удален' | RO: 'Defectiune: Ejectorul nu e in spate\\ E2.3 nu dispare' | ES: 'Error de funcionamiento: Eyector no está en la parte posterior , E1.13 no desaparece la señal' | PL: 'Nieprawidłowość:  Wyrzutnik nie jest z tyłu  , E1.13 Pozostało' | JA: 'エラー: エジェクタが後方に有りません 2.3\u3000未完了' | ZH: '故障: 弹射器不在后面 , E1.13 故障没有解除'
  622 = 'Reserve (r106_6)' | EN: 'Reserve (r106_6)' | DE: 'Reserve (r106_6)' | FR: 'Reserve (r106_6)' | HU: 'Reserve (r106_6)' | IT: 'Reserve (r106_6)' | RU: 'Reserve (r106_6)' | RO: 'Reserve (r106_6)' | ES: 'Reserve (r106_6)' | PL: 'Reserve (r106_6)' | JA: 'Reserve (r106_6)' | ZH: 'Reserve (r106_6)'
  623 = 'Wartungs-Zähler hat Vorwahl erreicht, weiter mit Reset' | EN: 'Maintenance counter preselection reached  (Continue with Reset)' | DE: 'Wartungs-Zähler hat Vorwahl erreicht, weiter mit Reset' | FR: 'Compteur maintenance a atteint présélection continuer avec Reset' | HU: 'Karbantartás-számláló elérte a beállított értéket tovább Reset-tel' | IT: 'Raggiunto valore cicli per manutenzione  (Continuare con RESET)' | RU: 'Счетчик обслуживания  код достигнут  продолжить с Reset' | RO: 'Numaratorul de intretinere\\ a realizat cantitatea preselectata\\ continua cu RESET' | ES: 'Preselección del contador de mantenimiento alcanzado  (Continuar con Reset)' | PL: 'Wstępnie wybrana ilość licznika obsługi została osiągnięta  (Kontynuacja poprzez przycisk Reset)' | JA: 'メンテナンスまでのカウンター (リセットで継続）' | ZH: '预设保养次数达到  (复位按钮继续)'
  624 = 'Stückzahl-Vorwahl erreicht (weiter mit Reset)' | EN: 'Quantity preselection reached (Continue with Reset)' | DE: 'Stückzahl-Vorwahl erreicht (weiter mit Reset)' | FR: 'Préselection nbre de pces atteint (continuer avec Reset)' | HU: 'Darabszám elérte a beállított értéket (tovább Reset-tel)' | IT: 'Raggiunta quantità pre-selezionata (Continuare con RESET)' | RU: 'Заданное кол-во достигнуто (продолжить c Reset)' | RO: 'Cantitatea preselectata realizata (continua cu RESET)' | ES: 'Cantidad preseleccionada alcanzada (Continuar con Reset)' | PL: 'Ilość wstępnie wybrana została osiągnięta (Kontynuacja poprzez przycisk Reset)' | JA: '設定数量達成 リセットで継続' | ZH: '预设总数到达 (复位按钮继续)'
  625 = 'Reserve (r107_1)'
  626 = 'Reserve (r107_2)'
  627 = 'Reserve (r107_3)'
  628 = 'Reserve (r107_4)'
  629 = 'Reserve (r107_5)'
  630 = 'Reserve (r107_6)'
  631 = 'Reserve (r107_7)'
   = ''
END_TEXTLIST

(* stored: Version 1.1.0.1, ProductVersion 3.1.4024.3
   TextList BetrAnzeigeListe: Id {ae46d11a-a98c-426e-8b75-ebbdf9c4c560} *)
